FUNCTION_BLOCK ButtonNO EXTENDS Button
VAR
	input AT %I* : BOOL;
END_VAR

PROPERTY IsPressed : BOOL
GET
IsPressed := input;
END_GET
END_PROPERTY

PROPERTY IsReleased : BOOL
GET
IsReleased := NOT input;
END_GET
END_PROPERTY

END_FUNCTION_BLOCK

(* stored: Version 1.1.0.1, ProductVersion 3.1.4024.12
   POU ButtonNO: Id {b503bddc-38ca-4d62-8359-601e5b924133}, SpecialFunc None
   Property IsPressed: Id {57f57dcd-341b-4652-a81c-264299f27931}
   Get Get: Id {268cd101-e03e-49a7-a012-5ca5da513eca}
   Property IsReleased: Id {8562a8f3-f686-4bc7-a4b1-85d9c6e8ecfc}
   Get Get: Id {c2677609-7d27-4eda-a2da-87b7ae7910de} *)
